TYPE HOLIDAY_DATA :
STRUCT
	NAME : STRING(30);
	DAY : SINT;
	MONTH : SINT;
	USE : SINT;
END_STRUCT
END_TYPE

(* stored: Version 1.1.0.1
   DUT HOLIDAY_DATA: Id {9d04fe60-c902-44da-9591-ef6f1eba49e9} *)
